Staubli VAL3: setStatus.pgx

public program setStatus(bool x_bStatus, string x_sId)
begin
  // change the BIT status
  saveInOut:dOutput[x_sId].dDio=x_bStatus
end
